FUNCTION_BLOCK JUnitResultFile IMPLEMENTS I_UnitTestResultFile
VAR
	Initialized, Write					: BOOL;
	XmlDomParser						: FB_XmlDomParser;
	RootNode, TestSuitesNode, TestSuite : SXmlNode;
	Path								: STRING;
END_VAR

METHOD AddTestCaseResult
VAR_INPUT
	Name			: STRING;
	Test			: STRING;
	Duration		: LREAL;
	FailtureMessage : STRING := '';
	FailtureType	: STRING := '';
	FailtureNote	: STRING := '';
END_VAR
IF NOT Initialized THEN
    RETURN;
END_IF
END_METHOD

METHOD AddTestSuite
VAR_INPUT
	Name	  : STRING;
	Tests	  : UDINT;
	Failtures : UDINT := 0;
	Errors	  : UDINT := 0;
	Skipped	  : UDINT := 0;
	Duration  : LREAL;
END_VAR
IF NOT Initialized THEN
	RETURN;
END_IF

TestSuite := XmlDomParser.AppendChild(TestSuitesNode,
									  'testsuite',
									  'TestSuite Core',
									  FALSE);
END_METHOD

METHOD Cyclic
XmlDomParser.SaveDocumentToFile(Path, Write);
END_METHOD

//FB_Init is always available implicitly and it is used primarily for initialization.

//The return value is not evaluated. For a specific influence, you can also declare the

//methods explicitly and provide additional code there with the standard initialization

//code. You can evaluate the return value.
METHOD FB_Init : BOOL
VAR_INPUT
	bInitRetains : BOOL; // TRUE: the retain variables are initialized (reset warm / reset cold)
	bInCopyCode	 : BOOL; // TRUE: the instance will be copied to the copy code afterward (online change)   
	Path		 : STRING;
END_VAR
THIS^.Path := Path;
END_METHOD

METHOD Initialize
VAR_INPUT
	ReInitialize : BOOL := FALSE;
END_VAR
IF Initialized AND NOT ReInitialize THEN
	RETURN;
END_IF

XmlDomParser.NewDocument();
RootNode	   := XmlDomParser.GetDocumentNode();
TestSuitesNode := XmlDomParser.AppendChild(RootNode,
										   'testsuites',
										   '',
										   FALSE);

Initialized := TRUE;
END_METHOD

METHOD SaveResult
IF NOT Initialized THEN
	RETURN;
END_IF

Write := TRUE;
END_METHOD

END_FUNCTION_BLOCK

(* stored: Version 1.1.0.1
   POU JUnitResultFile: Id {467a2f7d-ea77-463d-bccb-4ff68e52df26}, SpecialFunc None
   Method AddTestCaseResult: Id {fef2152d-9883-418e-81df-19425d45758e}
   Method AddTestSuite: Id {b9ed6143-3d62-40dc-ab57-7f199b7a8267}
   Method Cyclic: Id {4a8e3fe5-235e-4dba-86c7-512836695edb}
   Method FB_Init: Id {cf7f13e2-e0dc-4b72-817e-6e09f7f78b6d}
   Method Initialize: Id {23d2b239-3906-4cef-b04c-0fd9ab13f256}
   Method SaveResult: Id {24be214b-5fc2-42d3-8a34-ff3a2fc199dd} *)
